FUNCTION_BLOCK FB_Fenster_Ablaufsteuerung
VAR_IN_OUT
	Zustand			: ST_Fenster_Zustand;
	Stellwert		: ST_Fenster_Stellwert;
END_VAR
VAR_INPUT
	Steuerung		: ST_Fenster_Steuerung;
	Parameter		: ST_Fenster_Parameter;
END_VAR
VAR_OUTPUT
END_VAR
VAR
	Timer		: TON;
	E_Fenster_Zustand_Stellungwechsel10						: SINT;
	E_Fenster_Zustand_Stellungwechsel01						: SINT;
	E_Fenster_Zustand_Status_Stellungrueckmeldung0_Sperre	: SINT;
	E_Fenster_Zustand_Status_Stellungrueckmeldung0			: SINT;
	E_Fenster_Zustand_Status_Stellungrueckmeldung1_Sperre	: SINT;
	E_Fenster_Zustand_Status_Stellungrueckmeldung1			: SINT;
END_VAR

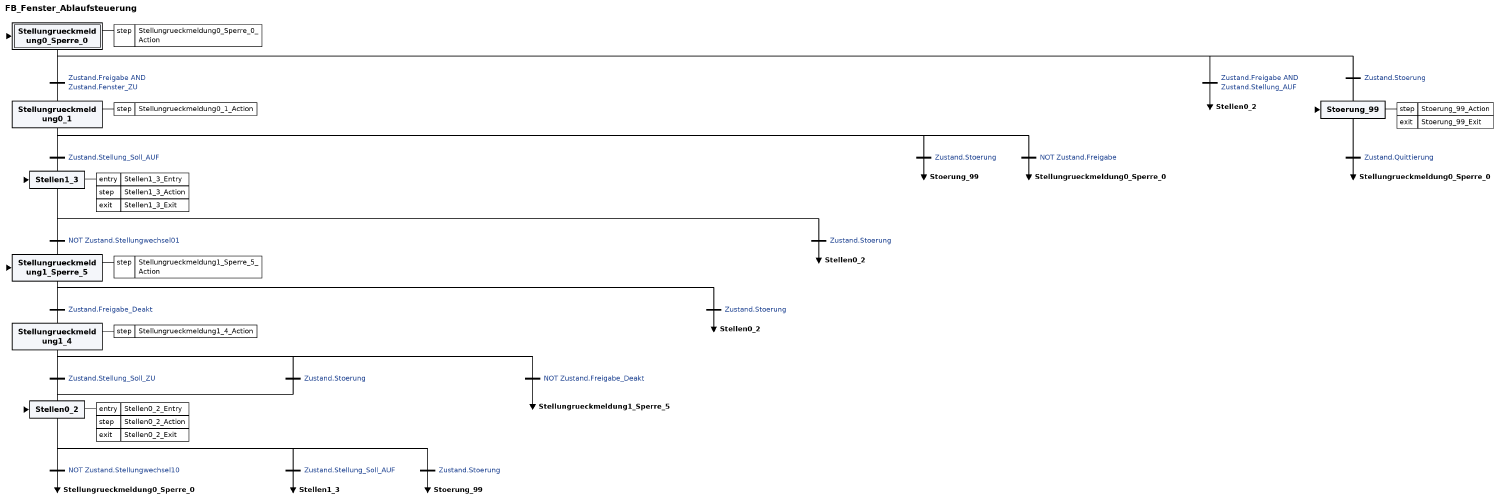
INITIAL_STEP Stellungrueckmeldung0_Sperre_0:
    Stellungrueckmeldung0_Sperre_0_Action(N);  // step action
END_STEP
TRANSITION FROM Stellungrueckmeldung0_Sperre_0 TO Stellungrueckmeldung0_1
    := Zustand.Freigabe AND Zustand.Fenster_ZU;
END_TRANSITION
TRANSITION FROM Stellungrueckmeldung0_Sperre_0 TO Stellen0_2
    := Zustand.Freigabe AND Zustand.Stellung_AUF;
END_TRANSITION
TRANSITION FROM Stellungrueckmeldung0_Sperre_0 TO Stoerung_99
    := Zustand.Stoerung;
END_TRANSITION
STEP Stoerung_99:
    Stoerung_99_Action(N);  // step action
    Stoerung_99_Exit(P0);  // exit action
END_STEP
TRANSITION FROM Stoerung_99 TO Stellungrueckmeldung0_Sperre_0
    := Zustand.Quittierung;
END_TRANSITION
STEP Stellungrueckmeldung0_1:
    Stellungrueckmeldung0_1_Action(N);  // step action
END_STEP
TRANSITION FROM Stellungrueckmeldung0_1 TO Stellen1_3
    := Zustand.Stellung_Soll_AUF;
END_TRANSITION
TRANSITION FROM Stellungrueckmeldung0_1 TO Stoerung_99
    := Zustand.Stoerung;
END_TRANSITION
TRANSITION FROM Stellungrueckmeldung0_1 TO Stellungrueckmeldung0_Sperre_0
    := NOT Zustand.Freigabe;
END_TRANSITION
STEP Stellen1_3:
    Stellen1_3_Entry(P1);  // entry action
    Stellen1_3_Action(N);  // step action
    Stellen1_3_Exit(P0);  // exit action
END_STEP
TRANSITION FROM Stellen1_3 TO Stellungrueckmeldung1_Sperre_5
    := NOT Zustand.Stellungwechsel01;
END_TRANSITION
TRANSITION FROM Stellen1_3 TO Stellen0_2
    := Zustand.Stoerung;
END_TRANSITION
STEP Stellungrueckmeldung1_Sperre_5:
    Stellungrueckmeldung1_Sperre_5_Action(N);  // step action
END_STEP
TRANSITION FROM Stellungrueckmeldung1_Sperre_5 TO Stellungrueckmeldung1_4
    := Zustand.Freigabe_Deakt;
END_TRANSITION
TRANSITION FROM Stellungrueckmeldung1_Sperre_5 TO Stellen0_2
    := Zustand.Stoerung;
END_TRANSITION
STEP Stellungrueckmeldung1_4:
    Stellungrueckmeldung1_4_Action(N);  // step action
END_STEP
TRANSITION FROM Stellungrueckmeldung1_4 TO Stellen0_2
    := Zustand.Stellung_Soll_ZU;
END_TRANSITION
TRANSITION FROM Stellungrueckmeldung1_4 TO Stellen0_2
    := Zustand.Stoerung;
END_TRANSITION
TRANSITION FROM Stellungrueckmeldung1_4 TO Stellungrueckmeldung1_Sperre_5
    := NOT Zustand.Freigabe_Deakt;
END_TRANSITION
STEP Stellen0_2:
    Stellen0_2_Entry(P1);  // entry action
    Stellen0_2_Action(N);  // step action
    Stellen0_2_Exit(P0);  // exit action
END_STEP
TRANSITION FROM Stellen0_2 TO Stellungrueckmeldung0_Sperre_0
    := NOT Zustand.Stellungwechsel10;
END_TRANSITION
TRANSITION FROM Stellen0_2 TO Stellen1_3
    := Zustand.Stellung_Soll_AUF;
END_TRANSITION
TRANSITION FROM Stellen0_2 TO Stoerung_99
    := Zustand.Stoerung;
END_TRANSITION

ACTION Stellen0_2_Action:
(* Nachlauf Timer starten *)
Timer( 	IN := Zustand.Stellungwechsel10,
		PT := DINT_TO_TIME(Parameter.Zeit_Stellen0),
);
Zustand.Stellungwechsel10	:= NOT Timer.Q;

(* Stellwert setzen *)
Stellwert.Fenster_AUF := FALSE;

(* Zustand setzen *)
Zustand.Status := E_Fenster_Zustand_Stellungwechsel10;
END_ACTION

ACTION Stellen0_2_Entry:
(* Reset Timer *)
Timer(IN := FALSE);
Zustand.Stellungwechsel10 := TRUE;
END_ACTION

ACTION Stellen0_2_Exit:
Zustand.Stellungwechsel10 := FALSE;
END_ACTION

ACTION Stellen1_3_Action:
(* Vorlaufzeit Timer starten *)
Timer( 	IN := Zustand.Stellungwechsel01,
		PT := DINT_TO_TIME(Parameter.Zeit_Stellen1),
);
Zustand.Stellungwechsel01	:= NOT Timer.Q;

(* Stellwert setzen *)
Stellwert.Fenster_AUF := TRUE;

(* Zustand setzen *)

Zustand.Status := E_Fenster_Zustand_Stellungwechsel01;
END_ACTION

ACTION Stellen1_3_Entry:
(* Reset Timer *)
Timer(IN := FALSE);
Zustand.Stellungwechsel01 := TRUE;
END_ACTION

ACTION Stellen1_3_Exit:
Zustand.Stellungwechsel01 := FALSE;
END_ACTION

ACTION Stellungrueckmeldung0_1_Action:
(* Stellwert setzen *)
Stellwert.Fenster_AUF := FALSE;
Zustand.Fenster_AUF := FALSE;

(* Zustand setzen *)
Zustand.Status := E_Fenster_Zustand_Status_Stellungrueckmeldung0;
END_ACTION

ACTION Stellungrueckmeldung0_Sperre_0_Action:
(* Stellwert setzen *)
Stellwert.Fenster_AUF:= FALSE;
(* Zustand setzen *)
Zustand.Fenster_ZU:= TRUE;

Zustand.Status := E_Fenster_Zustand_Status_Stellungrueckmeldung0_Sperre;
END_ACTION

ACTION Stellungrueckmeldung1_4_Action:
(* Stellwert setzen *)
Stellwert.Fenster_AUF := TRUE;

(* Zustand setzen *)
Zustand.Fenster_AUF := TRUE;
ZUstand.Fenster_ZU	:= FALSE;
Zustand.Status := E_Fenster_Zustand_Status_Stellungrueckmeldung1;
END_ACTION

ACTION Stellungrueckmeldung1_Sperre_5_Action:
(* Stellwert setzen *)
Stellwert.Fenster_AUF := TRUE;


(* Zustand setzen *)
Zustand.Fenster_AUF:= TRUE;
Zustand.Fenster_ZU:= FALSE;
Zustand.Status := E_Fenster_Zustand_Status_Stellungrueckmeldung1_Sperre;
END_ACTION

ACTION Stoerung_99_Action:
(* Stellwert setzen *)
Stellwert.Fenster_AUF := Zustand.Fenster_AUF;

(* Zustand setzen *)
Zustand.Stoerung := TRUE;
END_ACTION

ACTION Stoerung_99_Exit:
Zustand.Stoerung	:= FALSE;
END_ACTION

END_FUNCTION_BLOCK

(* stored: Version 1.1.0.1, ProductVersion 3.1.4024.9
   POU FB_Fenster_Ablaufsteuerung: Id {fd61d275-04b4-4f77-a578-76cfffc81fa0}, SpecialFunc None
   Action Stellen0_2_Action: Id {b1a04547-5f01-4054-baa9-1fa5e246d805}
   Action Stellen0_2_Entry: Id {a9dab52b-ae87-4111-8a6d-6f8d150faee0}
   Action Stellen0_2_Exit: Id {f3a26324-923d-45b6-b106-21b98960016c}
   Action Stellen1_3_Action: Id {e54f980f-beae-4e88-814c-b3a34290b676}
   Action Stellen1_3_Entry: Id {a30b1b3e-725f-4615-b2d7-6d221785e97e}
   Action Stellen1_3_Exit: Id {e904cd4d-1cb0-4bdb-9557-ee1ab76286db}
   Action Stellungrueckmeldung0_1_Action: Id {dc785ac4-b26b-40b3-b7b8-a1802187c97f}
   Action Stellungrueckmeldung0_Sperre_0_Action: Id {34a56c73-0d21-405d-af4b-0bc21e2e2e21}
   Action Stellungrueckmeldung1_4_Action: Id {2a11eee2-fccf-4085-b228-715c1cb4ff08}
   Action Stellungrueckmeldung1_Sperre_5_Action: Id {273025d1-6344-4dbc-9744-a638eab06165}
   Action Stoerung_99_Action: Id {bd4fb195-da0d-46ab-afc4-773344f944a9}
   Action Stoerung_99_Exit: Id {9c0ab693-f605-45be-9944-3a137bcadf0b} *)
